FUNCTION TryConvert_DWORD_TO_REAL : BOOL
VAR_INPUT
	in : DWORD;
	out : REFERENCE TO REAL;
END_VAR

out := DWORD_TO_REAL(in);
TryConvert_DWORD_TO_REAL := TRUE;

END_FUNCTION

(* stored: Version 1.1.0.1, ProductVersion 3.1.4024.12
   POU TryConvert_DWORD_TO_REAL: Id {bc86294d-63a0-46c3-af4f-cff546a679c1}, SpecialFunc None *)
